// Mitsubishi GX Works2 project: 12   PLC: FX3G

// task Task_01 (event TRUE, interval 0, priority 31): POU_01

PROGRAM POU_01
VAR
  wstep : INT;
  ton1 : TON;
  ton2 : TON;
END_VAR
IF M8002 THEN
	wstep := 0;
END_IF;

CASE wstep OF
	0:
		Y0 := FALSE;
		ton1(IN := M0, PT := T#1s);
		IF ton1.Q THEN
			ton1(IN := FALSE);
			wstep := 20;
		END_IF;
		
	20:
		ton1(IN := TRUE, PT := T#1s);
		Y0 := NOT ton1.Q;		
		
		IF NOT M0 THEN
			ton1(IN := FALSE);
			wstep := 21;
		END_IF;
	
	21:
		Y0 := TRUE;
		ton1(IN := TRUE, PT := T#1s);
		IF ton1.Q THEN
			ton1(IN := FALSE);
			wstep := 0;
		END_IF;

END_CASE;
END_PROGRAM
